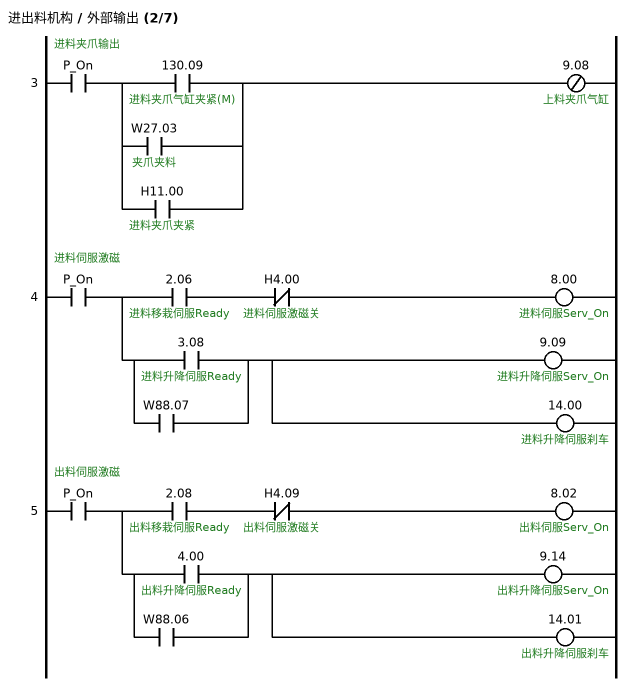
; [picture p120: 进出料机构 / 外部输出, rungs 3-5]
; rung 3: 进料夹爪输出
LD P_On
LD 130.09  ; 进料夹爪气缸夹紧(M)
OR W27.03  ; 夹爪夹料
OR H11.00  ; 进料夹爪夹紧
ANDLD
OUTNOT 9.08  ; 上料夹爪气缸
; rung 4: 进料伺服激磁
LD P_On
OUT TR0
AND 2.06  ; 进料移栽伺服Ready
ANDNOT H4.00  ; 进料伺服激磁关
OUT 8.00  ; 进料伺服Serv_On
LD TR0
LD 3.08  ; 进料升降伺服Ready
OR W88.07
ANDLD
OUT 9.09  ; 进料升降伺服Serv_On
OUT 14.00  ; 进料升降伺服刹车
; rung 5: 出料伺服激磁
LD P_On
OUT TR0
AND 2.08  ; 出料移栽伺服Ready
ANDNOT H4.09  ; 出料伺服激磁关
OUT 8.02  ; 出料伺服Serv_On
LD TR0
LD 4.00  ; 出料升降伺服Ready
OR W88.06
ANDLD
OUT 9.14  ; 出料升降伺服Serv_On
OUT 14.01  ; 出料升降伺服刹车

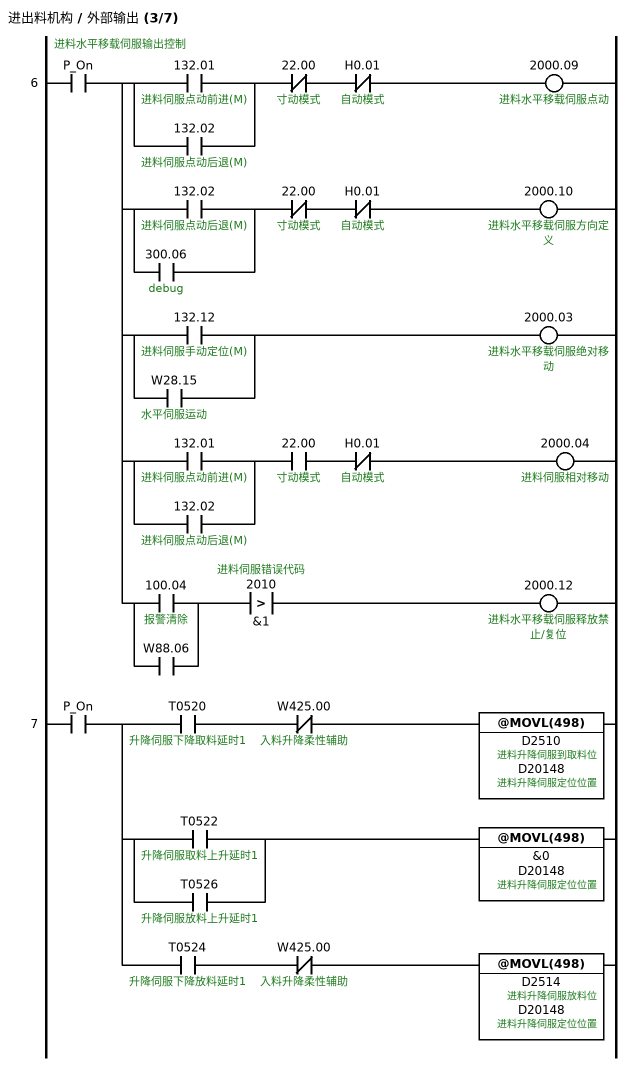
; rung 6: 进料水平移载伺服输出控制
LD P_On
OUT TR0
LD 132.01  ; 进料伺服点动前进(M)
OR 132.02  ; 进料伺服点动后退(M)
ANDLD
ANDNOT 22.00  ; 寸动模式
ANDNOT H0.01  ; 自动模式
OUT 2000.09  ; 进料水平移载伺服点动
LD TR0
LD 132.02  ; 进料伺服点动后退(M)
OR 300.06  ; debug
ANDLD
ANDNOT 22.00  ; 寸动模式
ANDNOT H0.01  ; 自动模式
OUT 2000.10  ; 进料水平移载伺服方向定义
LD TR0
LD 132.12  ; 进料伺服手动定位(M)
OR W28.15  ; 水平伺服运动
ANDLD
OUT 2000.03  ; 进料水平移载伺服绝对移动
LD TR0
LD 132.01  ; 进料伺服点动前进(M)
OR 132.02  ; 进料伺服点动后退(M)
ANDLD
AND 22.00  ; 寸动模式
ANDNOT H0.01  ; 自动模式
OUT 2000.04  ; 进料伺服相对移动
LD TR0
LD 100.04  ; 报警清除
OR W88.06
ANDLD
AND>(320) 2010 &1  ; 进料伺服错误代码
OUT 2000.12  ; 进料水平移载伺服释放禁止/复位
; rung 7
LD P_On
OUT TR0
AND T0520  ; 升降伺服下降取料延时1
ANDNOT W425.00  ; 入料升降柔性辅助
@MOVL(498) D2510 D20148  ; 进料升降伺服到取料位, 进料升降伺服定位位置
LD TR0
LD T0522  ; 升降伺服取料上升延时1
OR T0526  ; 升降伺服放料上升延时1
ANDLD
@MOVL(498) &0 D20148  ; 进料升降伺服定位位置
LD TR0
AND T0524  ; 升降伺服下降放料延时1
ANDNOT W425.00  ; 入料升降柔性辅助
@MOVL(498) D2514 D20148  ; 进料升降伺服放料位, 进料升降伺服定位位置

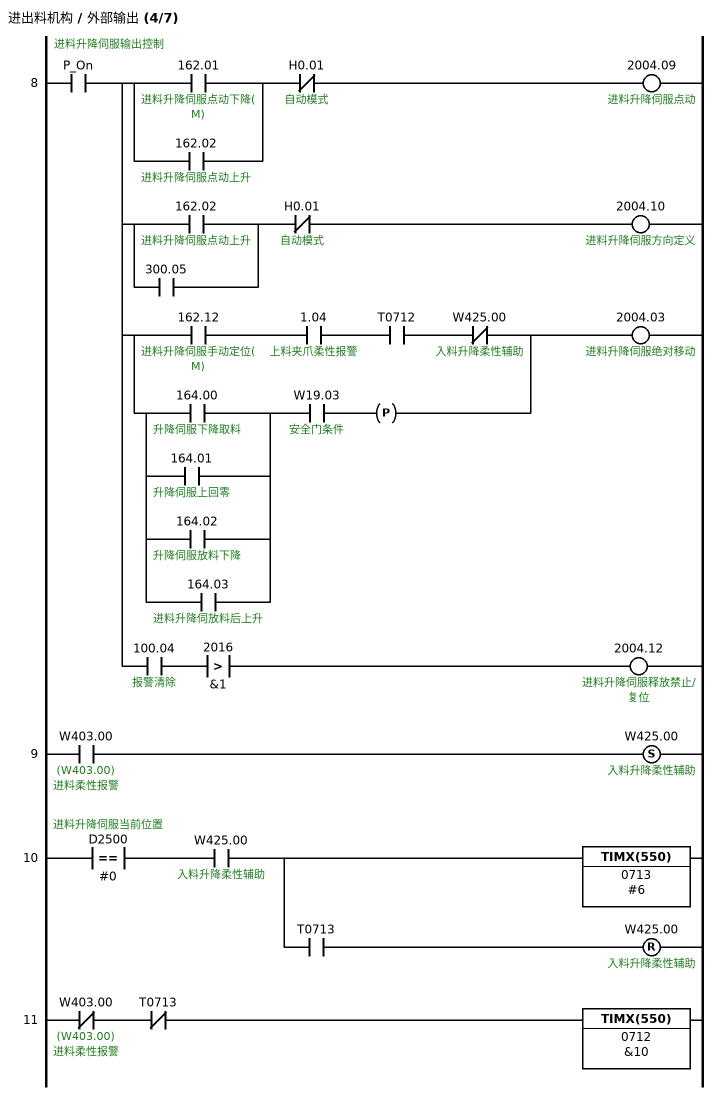
; rung 8: 进料升降伺服输出控制
LD P_On
OUT TR0
LD 162.01  ; 进料升降伺服点动下降(M)
OR 162.02  ; 进料升降伺服点动上升
ANDLD
ANDNOT H0.01  ; 自动模式
OUT 2004.09  ; 进料升降伺服点动
LD TR0
LD 162.02  ; 进料升降伺服点动上升
OR 300.05
ANDLD
ANDNOT H0.01  ; 自动模式
OUT 2004.10  ; 进料升降伺服方向定义
LD TR0
LD 162.12  ; 进料升降伺服手动定位(M)
AND 1.04  ; 上料夹爪柔性报警
AND T0712
ANDNOT W425.00  ; 入料升降柔性辅助
LD 164.00  ; 升降伺服下降取料
OR 164.01  ; 升降伺服上回零
OR 164.02  ; 升降伺服放料下降
OR 164.03  ; 进料升降伺放料后上升
AND W19.03  ; 安全门条件
UP(521)
ORLD
ANDLD
OUT 2004.03  ; 进料升降伺服绝对移动
LD TR0
AND 100.04  ; 报警清除
AND>(320) 2016 &1
OUT 2004.12  ; 进料升降伺服释放禁止/复位
; rung 9
LD W403.00  ; (W403.00) 进料柔性报警
SET W425.00  ; 入料升降柔性辅助
; rung 10
LD=L(301) D2500 #0  ; 进料升降伺服当前位置
AND W425.00  ; 入料升降柔性辅助
TIMX(550) 0713 #6
AND T0713
RSET W425.00  ; 入料升降柔性辅助
; rung 11
LDNOT W403.00  ; (W403.00) 进料柔性报警
ANDNOT T0713
TIMX(550) 0712 &10

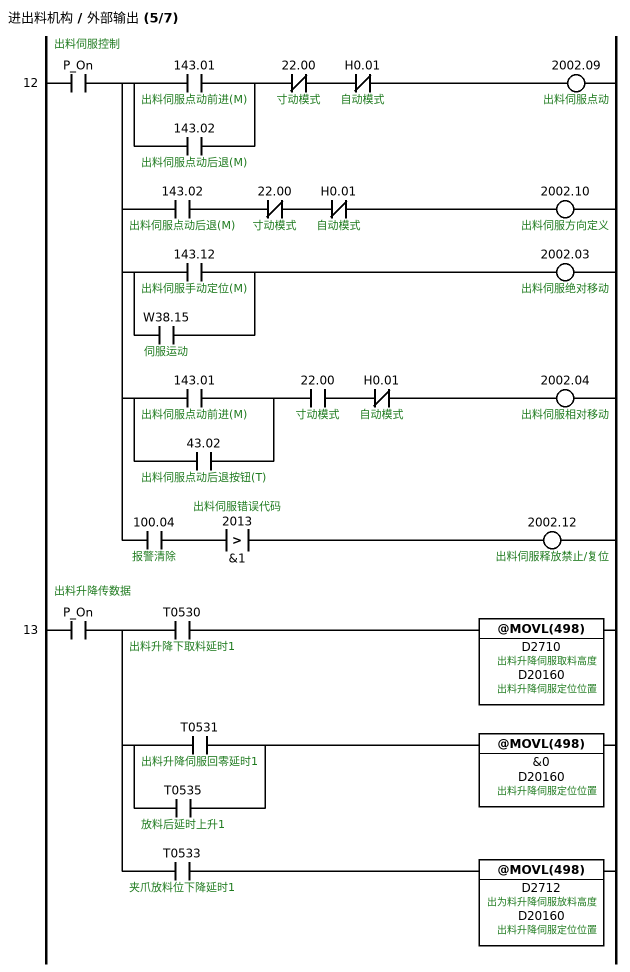
; rung 12: 出料伺服控制
LD P_On
OUT TR0
LD 143.01  ; 出料伺服点动前进(M)
OR 143.02  ; 出料伺服点动后退(M)
ANDLD
ANDNOT 22.00  ; 寸动模式
ANDNOT H0.01  ; 自动模式
OUT 2002.09  ; 出料伺服点动
LD TR0
AND 143.02  ; 出料伺服点动后退(M)
ANDNOT 22.00  ; 寸动模式
ANDNOT H0.01  ; 自动模式
OUT 2002.10  ; 出料伺服方向定义
LD TR0
LD 143.12  ; 出料伺服手动定位(M)
OR W38.15  ; 伺服运动
ANDLD
OUT 2002.03  ; 出料伺服绝对移动
LD TR0
LD 143.01  ; 出料伺服点动前进(M)
OR 43.02  ; 出料伺服点动后退按钮(T)
ANDLD
AND 22.00  ; 寸动模式
ANDNOT H0.01  ; 自动模式
OUT 2002.04  ; 出料伺服相对移动
LD TR0
AND 100.04  ; 报警清除
AND>(320) 2013 &1  ; 出料伺服错误代码
OUT 2002.12  ; 出料伺服释放禁止/复位
; rung 13: 出料升降传数据
LD P_On
OUT TR0
AND T0530  ; 出料升降下取料延时1
@MOVL(498) D2710 D20160  ; 出料升降伺服取料高度, 出料升降伺服定位位置
LD TR0
LD T0531  ; 出料升降伺服回零延时1
OR T0535  ; 放料后延时上升1
ANDLD
@MOVL(498) &0 D20160  ; 出料升降伺服定位位置
LD TR0
AND T0533  ; 夹爪放料位下降延时1
@MOVL(498) D2712 D20160  ; 出为料升降伺服放料高度, 出料升降伺服定位位置

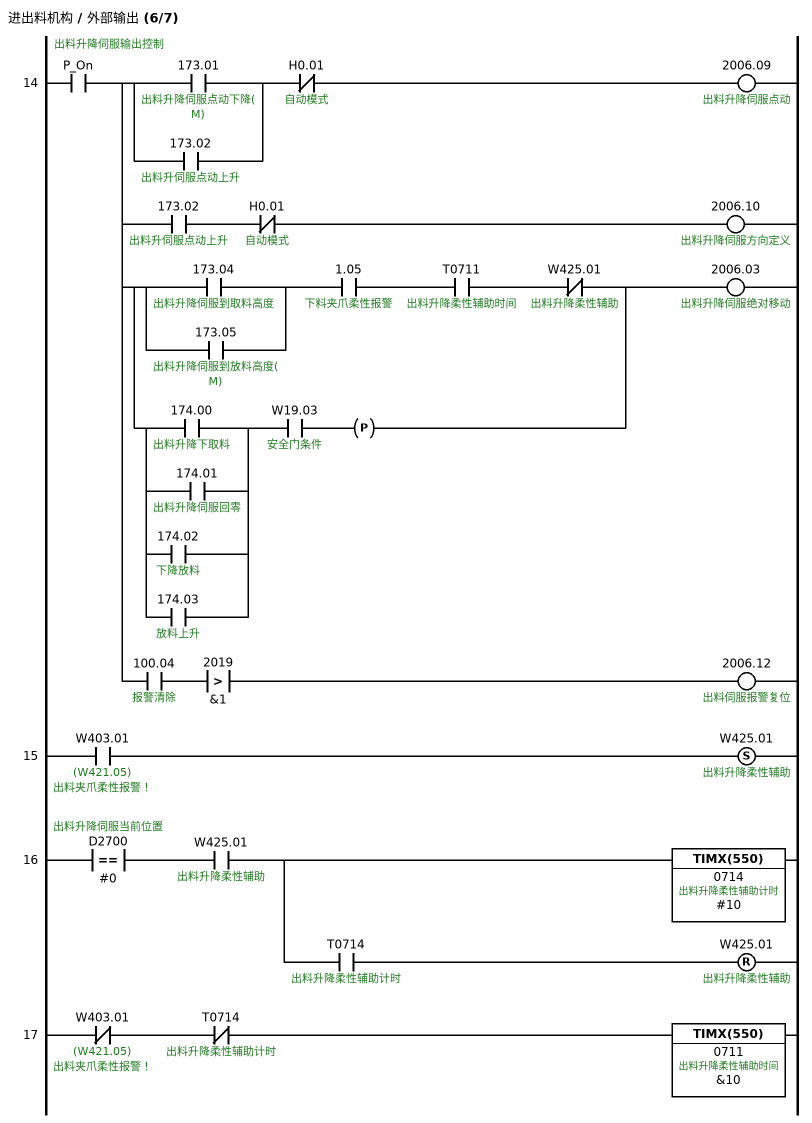
; rung 14: 出料升降伺服输出控制
LD P_On
OUT TR0
LD 173.01  ; 出料升降伺服点动下降(M)
OR 173.02  ; 出料升伺服点动上升
ANDLD
ANDNOT H0.01  ; 自动模式
OUT 2006.09  ; 出料升降伺服点动
LD TR0
AND 173.02  ; 出料升伺服点动上升
ANDNOT H0.01  ; 自动模式
OUT 2006.10  ; 出料升降伺服方向定义
LD TR0
LD 173.04  ; 出料升降伺服到取料高度
OR 173.05  ; 出料升降伺服到放料高度(M)
AND 1.05  ; 下料夹爪柔性报警
AND T0711  ; 出料升降柔性辅助时间
ANDNOT W425.01  ; 出料升降柔性辅助
LD 174.00  ; 出料升降下取料
OR 174.01  ; 出料升降伺服回零
OR 174.02  ; 下降放料
OR 174.03  ; 放料上升
AND W19.03  ; 安全门条件
UP(521)
ORLD
ANDLD
OUT 2006.03  ; 出料升降伺服绝对移动
LD TR0
AND 100.04  ; 报警清除
AND>(320) 2019 &1
OUT 2006.12  ; 出料伺服报警复位
; rung 15
LD W403.01  ; (W421.05) 出料夹爪柔性报警！
SET W425.01  ; 出料升降柔性辅助
; rung 16
LD=L(301) D2700 #0  ; 出料升降伺服当前位置
AND W425.01  ; 出料升降柔性辅助
TIMX(550) 0714 #10  ; 出料升降柔性辅助计时
AND T0714  ; 出料升降柔性辅助计时
RSET W425.01  ; 出料升降柔性辅助
; rung 17
LDNOT W403.01  ; (W421.05) 出料夹爪柔性报警！
ANDNOT T0714  ; 出料升降柔性辅助计时
TIMX(550) 0711 &10  ; 出料升降柔性辅助时间

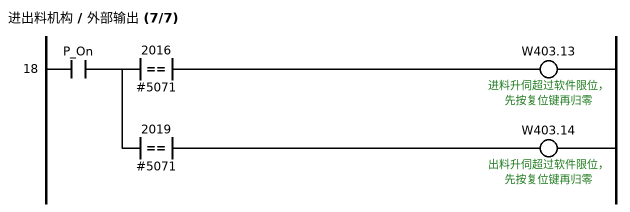
; rung 18
LD P_On
OUT TR0
AND=(300) 2016 #5071
OUT W403.13  ; 进料升伺超过软件限位，先按复位键再归零
LD TR0
AND=(300) 2019 #5071
OUT W403.14  ; 出料升伺超过软件限位，先按复位键再归零

### Section 指示灯

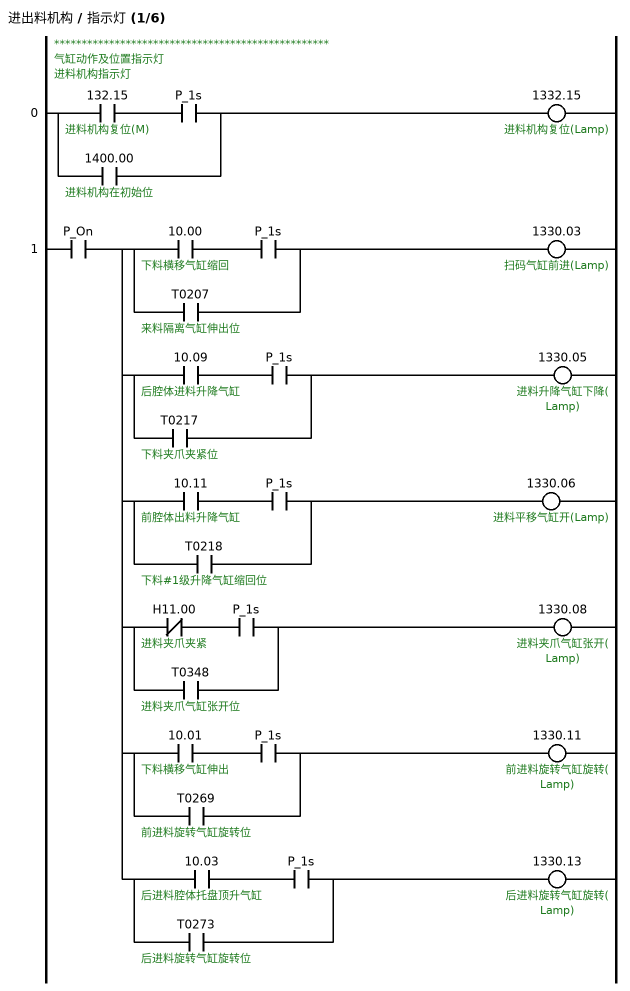
; rung 0: ************************************************** / 气缸动作及位置指示灯 / 进料机构指示灯
LD 132.15  ; 进料机构复位(M)
AND P_1s
OR 1400.00  ; 进料机构在初始位
OUT 1332.15  ; 进料机构复位(Lamp)
; rung 1
LD P_On
OUT TR0
LD 10.00  ; 下料横移气缸缩回
AND P_1s
OR T0207  ; 来料隔离气缸伸出位
ANDLD
OUT 1330.03  ; 扫码气缸前进(Lamp)
LD TR0
LD 10.09  ; 后腔体进料升降气缸
AND P_1s
OR T0217  ; 下料夹爪夹紧位
ANDLD
OUT 1330.05  ; 进料升降气缸下降(Lamp)
LD TR0
LD 10.11  ; 前腔体出料升降气缸
AND P_1s
OR T0218  ; 下料#1级升降气缸缩回位
ANDLD
OUT 1330.06  ; 进料平移气缸开(Lamp)
LD TR0
LDNOT H11.00  ; 进料夹爪夹紧
AND P_1s
OR T0348  ; 进料夹爪气缸张开位
ANDLD
OUT 1330.08  ; 进料夹爪气缸张开(Lamp)
LD TR0
LD 10.01  ; 下料横移气缸伸出
AND P_1s
OR T0269  ; 前进料旋转气缸旋转位
ANDLD
OUT 1330.11  ; 前进料旋转气缸旋转(Lamp)
LD TR0
LD 10.03  ; 后进料腔体托盘顶升气缸
AND P_1s
OR T0273  ; 后进料旋转气缸旋转位
ANDLD
OUT 1330.13  ; 后进料旋转气缸旋转(Lamp)

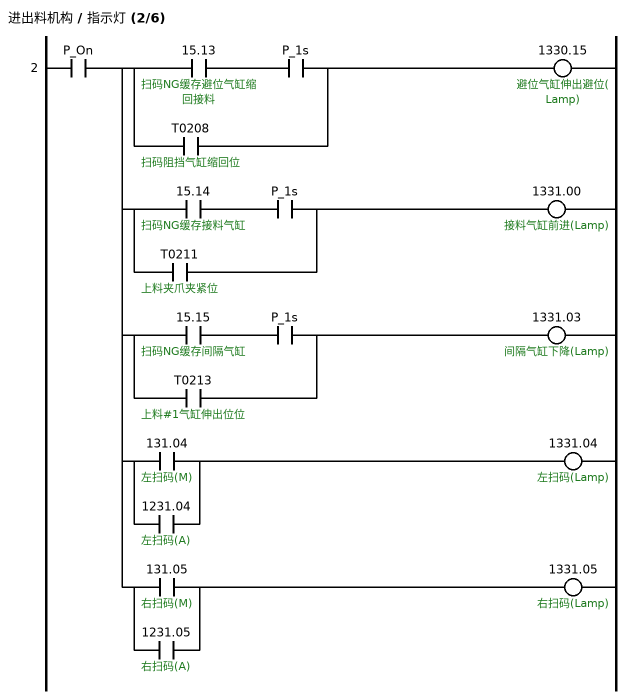
; rung 2
LD P_On
OUT TR0
LD 15.13  ; 扫码NG缓存避位气缸缩回接料
AND P_1s
OR T0208  ; 扫码阻挡气缸缩回位
ANDLD
OUT 1330.15  ; 避位气缸伸出避位(Lamp)
LD TR0
LD 15.14  ; 扫码NG缓存接料气缸
AND P_1s
OR T0211  ; 上料夹爪夹紧位
ANDLD
OUT 1331.00  ; 接料气缸前进(Lamp)
LD TR0
LD 15.15  ; 扫码NG缓存间隔气缸
AND P_1s
OR T0213  ; 上料#1气缸伸出位位
ANDLD
OUT 1331.03  ; 间隔气缸下降(Lamp)
LD TR0
LD 131.04  ; 左扫码(M)
OR 1231.04  ; 左扫码(A)
ANDLD
OUT 1331.04  ; 左扫码(Lamp)
LD TR0
LD 131.05  ; 右扫码(M)
OR 1231.05  ; 右扫码(A)
ANDLD
OUT 1331.05  ; 右扫码(Lamp)

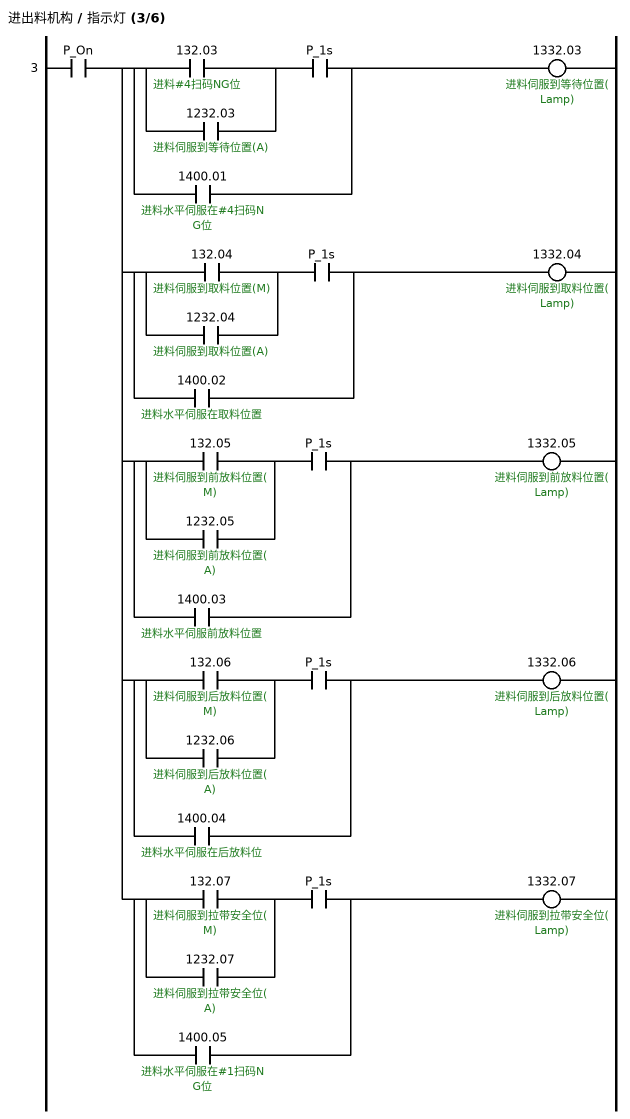
; rung 3
LD P_On
OUT TR0
LD 132.03  ; 进料#4扫码NG位
OR 1232.03  ; 进料伺服到等待位置(A)
AND P_1s
OR 1400.01  ; 进料水平伺服在#4扫码NG位
ANDLD
OUT 1332.03  ; 进料伺服到等待位置(Lamp)
LD TR0
LD 132.04  ; 进料伺服到取料位置(M)
OR 1232.04  ; 进料伺服到取料位置(A)
AND P_1s
OR 1400.02  ; 进料水平伺服在取料位置
ANDLD
OUT 1332.04  ; 进料伺服到取料位置(Lamp)
LD TR0
LD 132.05  ; 进料伺服到前放料位置(M)
OR 1232.05  ; 进料伺服到前放料位置(A)
AND P_1s
OR 1400.03  ; 进料水平伺服前放料位置
ANDLD
OUT 1332.05  ; 进料伺服到前放料位置(Lamp)
LD TR0
LD 132.06  ; 进料伺服到后放料位置(M)
OR 1232.06  ; 进料伺服到后放料位置(A)
AND P_1s
OR 1400.04  ; 进料水平伺服在后放料位
ANDLD
OUT 1332.06  ; 进料伺服到后放料位置(Lamp)
LD TR0
LD 132.07  ; 进料伺服到拉带安全位(M)
OR 1232.07  ; 进料伺服到拉带安全位(A)
AND P_1s
OR 1400.05  ; 进料水平伺服在#1扫码NG位
ANDLD
OUT 1332.07  ; 进料伺服到拉带安全位(Lamp)

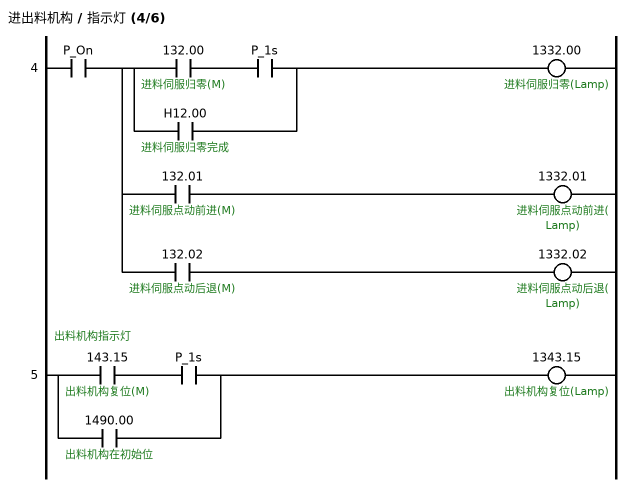
; rung 4
LD P_On
OUT TR0
LD 132.00  ; 进料伺服归零(M)
AND P_1s
OR H12.00  ; 进料伺服归零完成
ANDLD
OUT 1332.00  ; 进料伺服归零(Lamp)
LD TR0
AND 132.01  ; 进料伺服点动前进(M)
OUT 1332.01  ; 进料伺服点动前进(Lamp)
LD TR0
AND 132.02  ; 进料伺服点动后退(M)
OUT 1332.02  ; 进料伺服点动后退(Lamp)
; rung 5: 出料机构指示灯
LD 143.15  ; 出料机构复位(M)
AND P_1s
OR 1490.00  ; 出料机构在初始位
OUT 1343.15  ; 出料机构复位(Lamp)

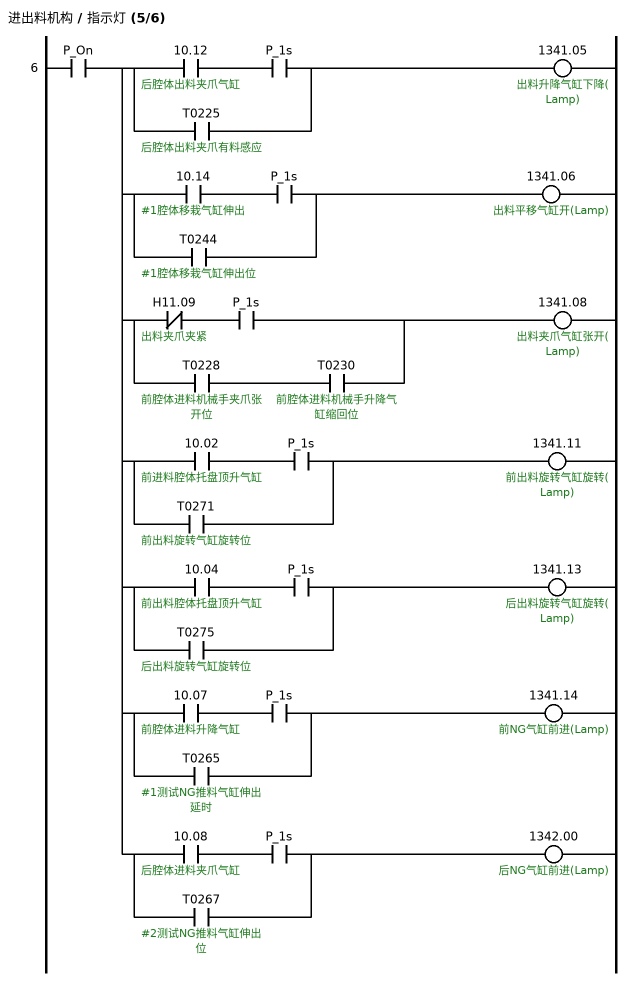
; rung 6
LD P_On
OUT TR0
LD 10.12  ; 后腔体出料夹爪气缸
AND P_1s
OR T0225  ; 后腔体出料夹爪有料感应
ANDLD
OUT 1341.05  ; 出料升降气缸下降(Lamp)
LD TR0
LD 10.14  ; #1腔体移栽气缸伸出
AND P_1s
OR T0244  ; #1腔体移栽气缸伸出位
ANDLD
OUT 1341.06  ; 出料平移气缸开(Lamp)
LD TR0
LDNOT H11.09  ; 出料夹爪夹紧
AND P_1s
LD T0228  ; 前腔体进料机械手夹爪张开位
AND T0230  ; 前腔体进料机械手升降气缸缩回位
ORLD
ANDLD
OUT 1341.08  ; 出料夹爪气缸张开(Lamp)
LD TR0
LD 10.02  ; 前进料腔体托盘顶升气缸
AND P_1s
OR T0271  ; 前出料旋转气缸旋转位
ANDLD
OUT 1341.11  ; 前出料旋转气缸旋转(Lamp)
LD TR0
LD 10.04  ; 前出料腔体托盘顶升气缸
AND P_1s
OR T0275  ; 后出料旋转气缸旋转位
ANDLD
OUT 1341.13  ; 后出料旋转气缸旋转(Lamp)
LD TR0
LD 10.07  ; 前腔体进料升降气缸
AND P_1s
OR T0265  ; #1测试NG推料气缸伸出延时
ANDLD
OUT 1341.14  ; 前NG气缸前进(Lamp)
LD TR0
LD 10.08  ; 后腔体进料夹爪气缸
AND P_1s
OR T0267  ; #2测试NG推料气缸伸出位
ANDLD
OUT 1342.00  ; 后NG气缸前进(Lamp)

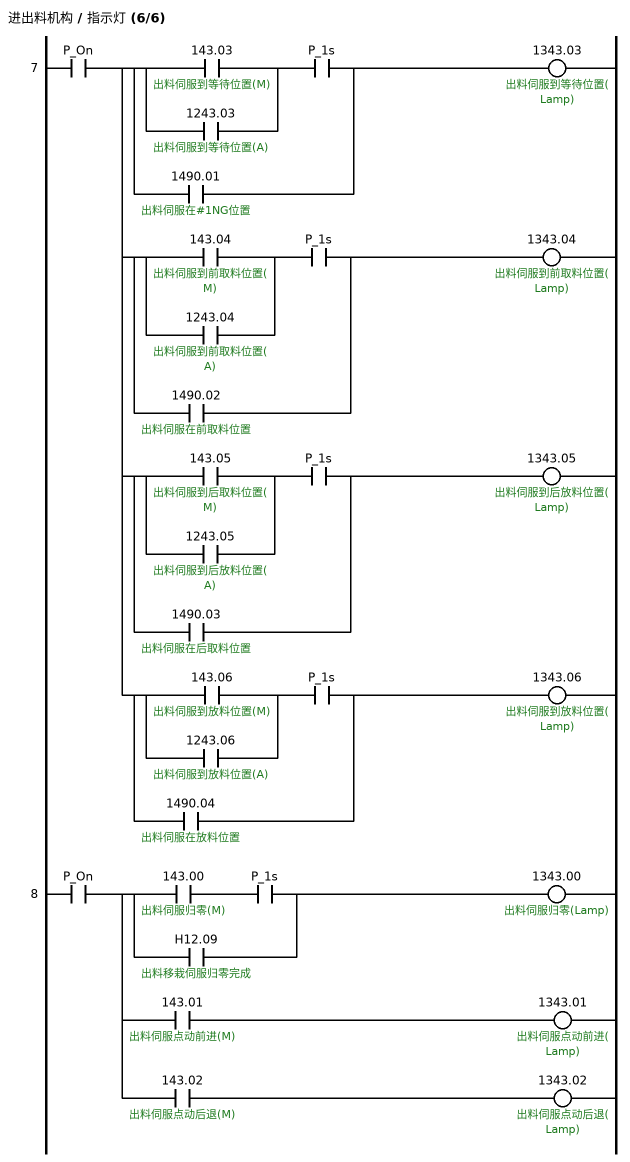
; rung 7
LD P_On
OUT TR0
LD 143.03  ; 出料伺服到等待位置(M)
OR 1243.03  ; 出料伺服到等待位置(A)
AND P_1s
OR 1490.01  ; 出料伺服在#1NG位置
ANDLD
OUT 1343.03  ; 出料伺服到等待位置(Lamp)
LD TR0
LD 143.04  ; 出料伺服到前取料位置(M)
OR 1243.04  ; 出料伺服到前取料位置(A)
AND P_1s
OR 1490.02  ; 出料伺服在前取料位置
ANDLD
OUT 1343.04  ; 出料伺服到前取料位置(Lamp)
LD TR0
LD 143.05  ; 出料伺服到后取料位置(M)
OR 1243.05  ; 出料伺服到后放料位置(A)
AND P_1s
OR 1490.03  ; 出料伺服在后取料位置
ANDLD
OUT 1343.05  ; 出料伺服到后放料位置(Lamp)
LD TR0
LD 143.06  ; 出料伺服到放料位置(M)
OR 1243.06  ; 出料伺服到放料位置(A)
AND P_1s
OR 1490.04  ; 出料伺服在放料位置
ANDLD
OUT 1343.06  ; 出料伺服到放料位置(Lamp)
; rung 8
LD P_On
OUT TR0
LD 143.00  ; 出料伺服归零(M)
AND P_1s
OR H12.09  ; 出料移栽伺服归零完成
ANDLD
OUT 1343.00  ; 出料伺服归零(Lamp)
LD TR0
AND 143.01  ; 出料伺服点动前进(M)
OUT 1343.01  ; 出料伺服点动前进(Lamp)
LD TR0
AND 143.02  ; 出料伺服点动后退(M)
OUT 1343.02  ; 出料伺服点动后退(Lamp)

### Section END
; rung 0
END(001)

## Program 前上料机构 (cyclic task 2)

### Section Main

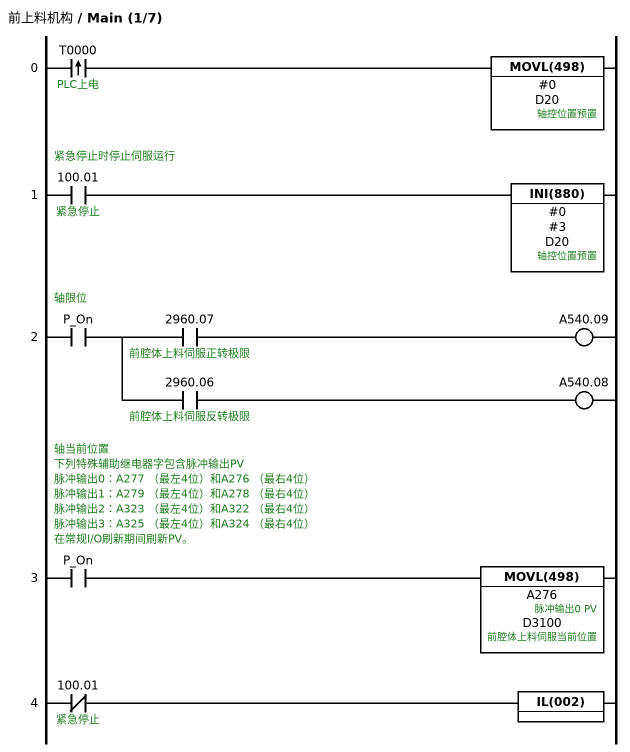
; rung 0
@LD T0000  ; PLC上电
MOVL(498) #0 D20  ; 轴控位置预置
; rung 1: 紧急停止时停止伺服运行
LD 100.01  ; 紧急停止
INI(880) #0 #3 D20  ; 轴控位置预置
; rung 2: 轴限位
LD P_On
OUT TR0
AND 2960.07  ; 前腔体上料伺服正转极限
OUT A540.09
LD TR0
AND 2960.06  ; 前腔体上料伺服反转极限
OUT A540.08
; rung 3: 轴当前位置 / 下列特殊辅助继电器字包含脉冲输出PV / 脉冲输出0：A277 （最左4位）和A276 （最右4位） / 脉冲输出1：A279 （最左4位）和A278 （最右4位） / 脉冲输出2：A323 （最左4位）和A322 （最右4位） / 脉冲输出3：A325 （最左4位）和A324 （最右4位） / 在常规I/O刷新期间刷新PV。
LD P_On
MOVL(498) A276 D3100  ; 脉冲输出0 PV, 前腔体上料伺服当前位置
; rung 4
LDNOT 100.01  ; 紧急停止
IL(002)

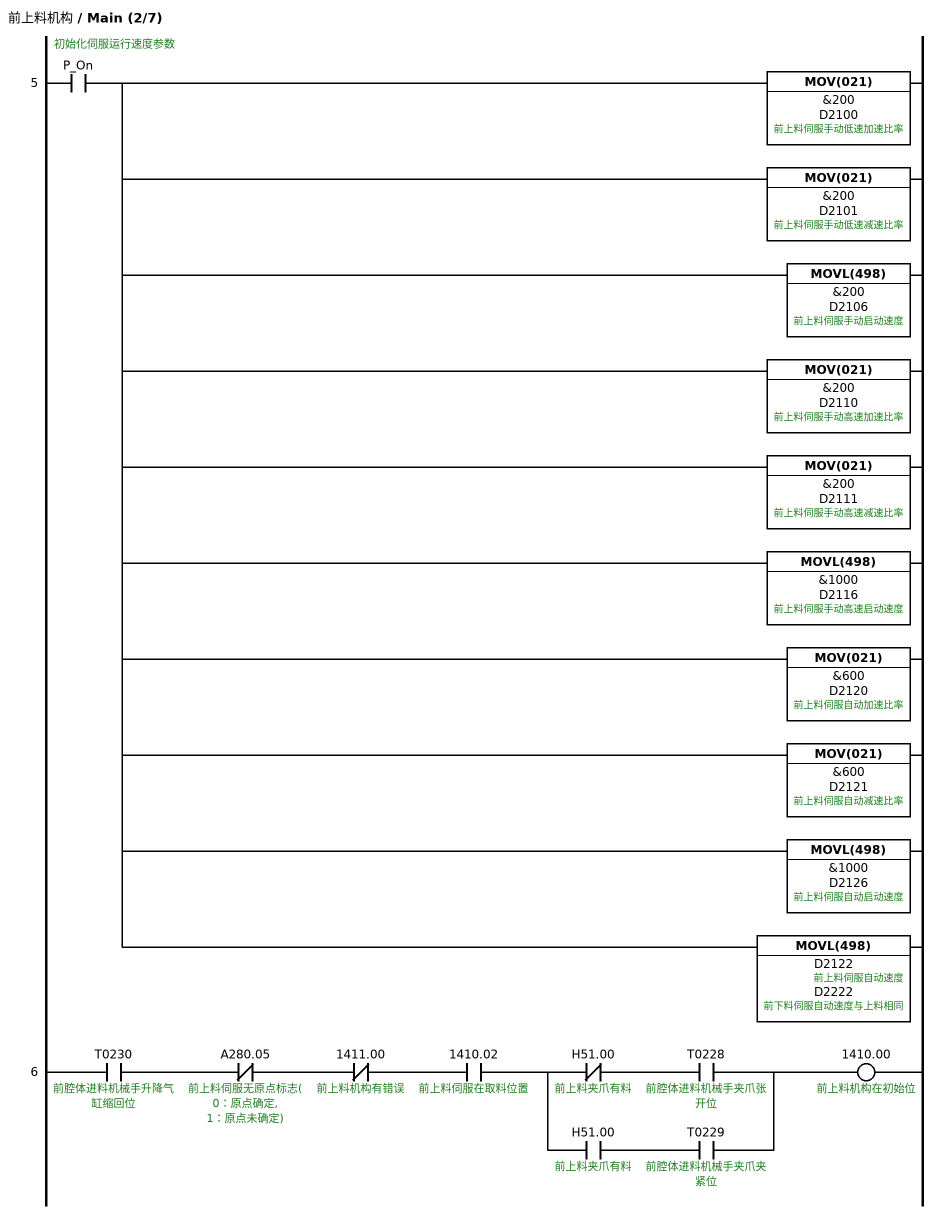
; rung 5: 初始化伺服运行速度参数
LD P_On
MOV(021) &200 D2100  ; 前上料伺服手动低速加速比率
MOV(021) &200 D2101  ; 前上料伺服手动低速减速比率
MOVL(498) &200 D2106  ; 前上料伺服手动启动速度
MOV(021) &200 D2110  ; 前上料伺服手动高速加速比率
MOV(021) &200 D2111  ; 前上料伺服手动高速减速比率
MOVL(498) &1000 D2116  ; 前上料伺服手动高速启动速度
MOV(021) &600 D2120  ; 前上料伺服自动加速比率
MOV(021) &600 D2121  ; 前上料伺服自动减速比率
MOVL(498) &1000 D2126  ; 前上料伺服自动启动速度
MOVL(498) D2122 D2222  ; 前上料伺服自动速度, 前下料伺服自动速度与上料相同
; rung 6
LD T0230  ; 前腔体进料机械手升降气缸缩回位
ANDNOT A280.05  ; 前上料伺服无原点标志(0：原点确定,1：原点未确定)
ANDNOT 1411.00  ; 前上料机构有错误
AND 1410.02  ; 前上料伺服在取料位置
LDNOT H51.00  ; 前上料夹爪有料
AND T0228  ; 前腔体进料机械手夹爪张开位
LD H51.00  ; 前上料夹爪有料
AND T0229  ; 前腔体进料机械手夹爪夹紧位
ORLD
ANDLD
OUT 1410.00  ; 前上料机构在初始位

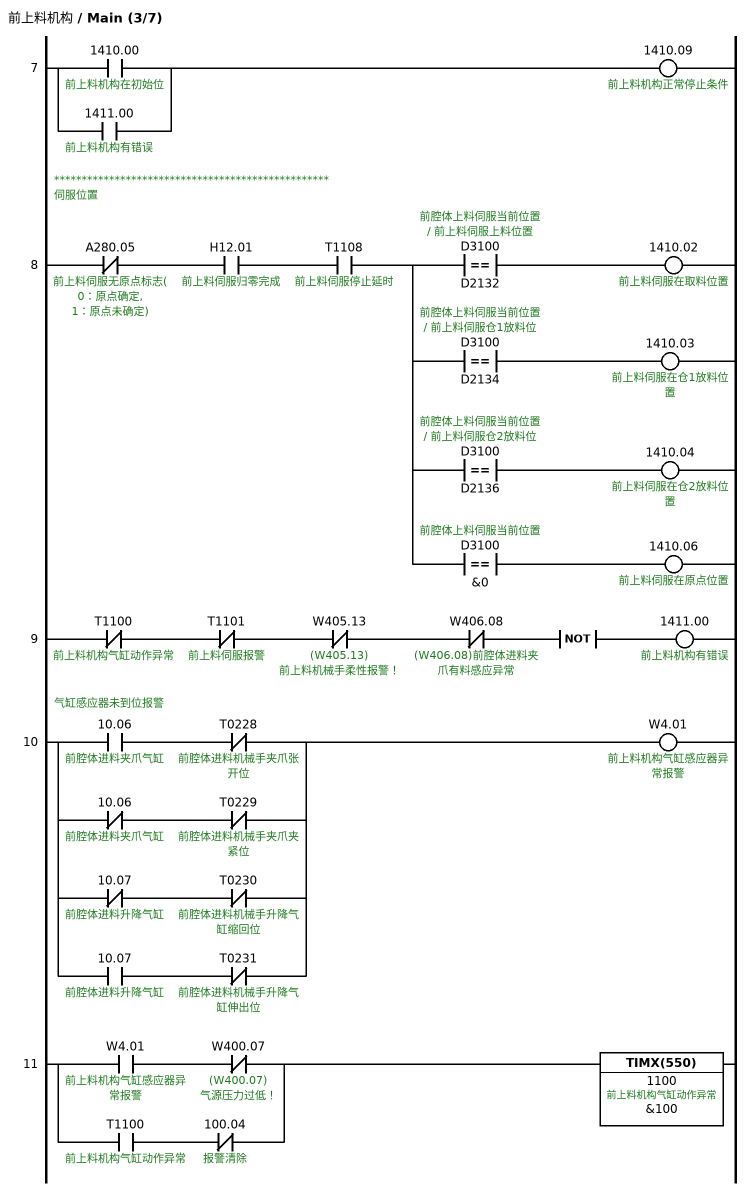
; rung 7
LD 1410.00  ; 前上料机构在初始位
OR 1411.00  ; 前上料机构有错误
OUT 1410.09  ; 前上料机构正常停止条件
; rung 8: ************************************************** / 伺服位置
LDNOT A280.05  ; 前上料伺服无原点标志(0：原点确定,1：原点未确定)
AND H12.01  ; 前上料伺服归零完成
AND T1108  ; 前上料伺服停止延时
OUT TR0
AND=SL(303) D3100 D2132  ; 前腔体上料伺服当前位置, 前上料伺服上料位置
OUT 1410.02  ; 前上料伺服在取料位置
LD TR0
AND=SL(303) D3100 D2134  ; 前腔体上料伺服当前位置, 前上料伺服仓1放料位
OUT 1410.03  ; 前上料伺服在仓1放料位置
LD TR0
AND=SL(303) D3100 D2136  ; 前腔体上料伺服当前位置, 前上料伺服仓2放料位
OUT 1410.04  ; 前上料伺服在仓2放料位置
LD TR0
AND=SL(303) D3100 &0  ; 前腔体上料伺服当前位置
OUT 1410.06  ; 前上料伺服在原点位置
; rung 9
LDNOT T1100  ; 前上料机构气缸动作异常
ANDNOT T1101  ; 前上料伺服报警
ANDNOT W405.13  ; (W405.13) 前上料机械手柔性报警！
ANDNOT W406.08  ; (W406.08)前腔体进料夹爪有料感应异常
NOT(520)
OUT 1411.00  ; 前上料机构有错误
; rung 10: 气缸感应器未到位报警
LD 10.06  ; 前腔体进料夹爪气缸
ANDNOT T0228  ; 前腔体进料机械手夹爪张开位
LDNOT 10.06  ; 前腔体进料夹爪气缸
ANDNOT T0229  ; 前腔体进料机械手夹爪夹紧位
ORLD
LDNOT 10.07  ; 前腔体进料升降气缸
ANDNOT T0230  ; 前腔体进料机械手升降气缸缩回位
ORLD
LD 10.07  ; 前腔体进料升降气缸
ANDNOT T0231  ; 前腔体进料机械手升降气缸伸出位
ORLD
OUT W4.01  ; 前上料机构气缸感应器异常报警
; rung 11
LD W4.01  ; 前上料机构气缸感应器异常报警
ANDNOT W400.07  ; (W400.07) 气源压力过低！
LD T1100  ; 前上料机构气缸动作异常
ANDNOT 100.04  ; 报警清除
ORLD
TIMX(550) 1100 &100  ; 前上料机构气缸动作异常

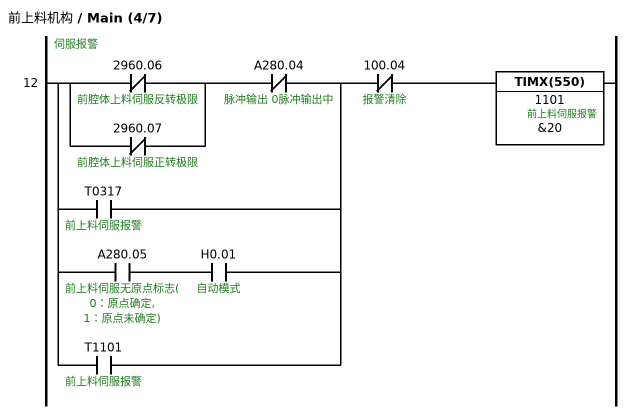
; rung 12: 伺服报警
LDNOT 2960.06  ; 前腔体上料伺服反转极限
ORNOT 2960.07  ; 前腔体上料伺服正转极限
ANDNOT A280.04  ; 脉冲输出 0脉冲输出中
OR T0317  ; 前上料伺服报警
LD A280.05  ; 前上料伺服无原点标志(0：原点确定,1：原点未确定)
AND H0.01  ; 自动模式
ORLD
OR T1101  ; 前上料伺服报警
ANDNOT 100.04  ; 报警清除
TIMX(550) 1101 &20  ; 前上料伺服报警

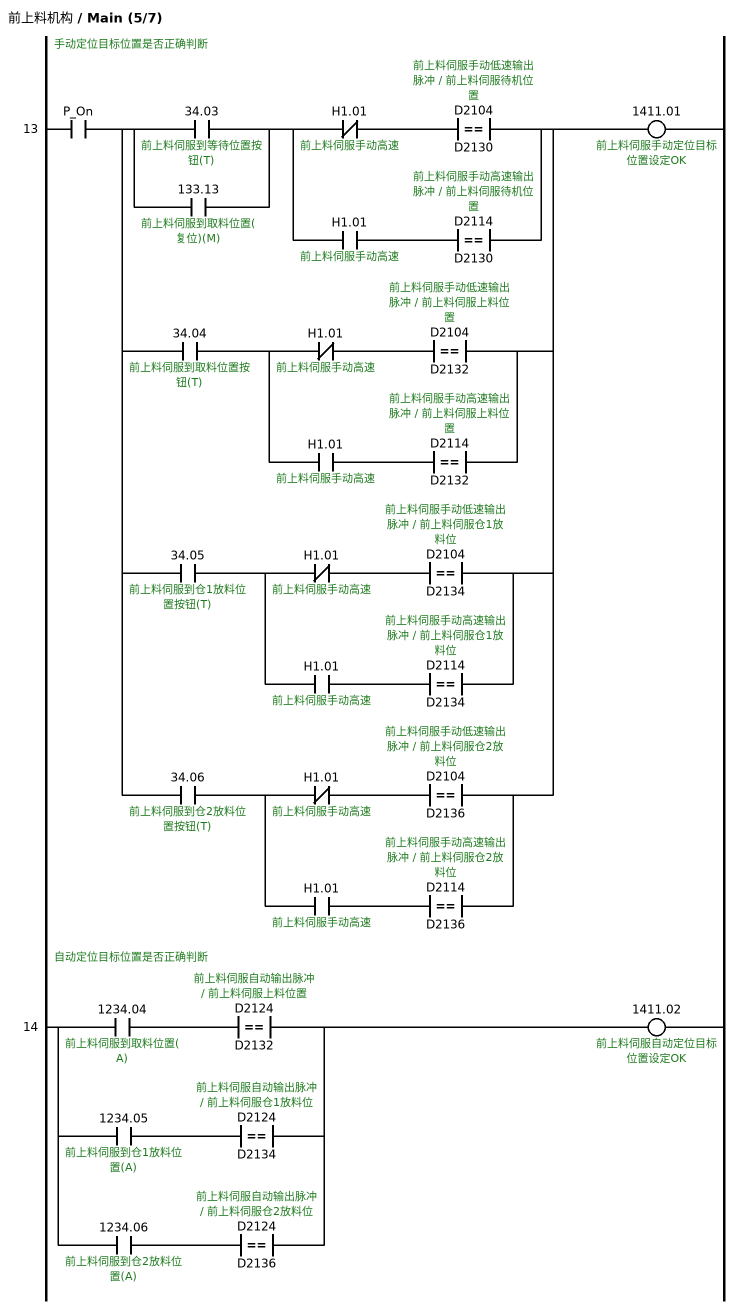
; rung 13: 手动定位目标位置是否正确判断
LD P_On
LD 34.03  ; 前上料伺服到等待位置按钮(T)
OR 133.13  ; 前上料伺服到取料位置(复位)(M)
LDNOT H1.01  ; 前上料伺服手动高速
AND=SL(303) D2104 D2130  ; 前上料伺服手动低速输出脉冲, 前上料伺服待机位置
LD H1.01  ; 前上料伺服手动高速
AND=SL(303) D2114 D2130  ; 前上料伺服手动高速输出脉冲, 前上料伺服待机位置
ORLD
ANDLD
LD 34.04  ; 前上料伺服到取料位置按钮(T)
LDNOT H1.01  ; 前上料伺服手动高速
AND=SL(303) D2104 D2132  ; 前上料伺服手动低速输出脉冲, 前上料伺服上料位置
LD H1.01  ; 前上料伺服手动高速
AND=SL(303) D2114 D2132  ; 前上料伺服手动高速输出脉冲, 前上料伺服上料位置
ORLD
ANDLD
ORLD
LD 34.05  ; 前上料伺服到仓1放料位置按钮(T)
LDNOT H1.01  ; 前上料伺服手动高速
AND=SL(303) D2104 D2134  ; 前上料伺服手动低速输出脉冲, 前上料伺服仓1放料位
LD H1.01  ; 前上料伺服手动高速
AND=SL(303) D2114 D2134  ; 前上料伺服手动高速输出脉冲, 前上料伺服仓1放料位
ORLD
ANDLD
ORLD
LD 34.06  ; 前上料伺服到仓2放料位置按钮(T)
LDNOT H1.01  ; 前上料伺服手动高速
AND=SL(303) D2104 D2136  ; 前上料伺服手动低速输出脉冲, 前上料伺服仓2放料位
LD H1.01  ; 前上料伺服手动高速
AND=SL(303) D2114 D2136  ; 前上料伺服手动高速输出脉冲, 前上料伺服仓2放料位
ORLD
ANDLD
ORLD
ANDLD
OUT 1411.01  ; 前上料伺服手动定位目标位置设定OK
; rung 14: 自动定位目标位置是否正确判断
LD 1234.04  ; 前上料伺服到取料位置(A)
AND=SL(303) D2124 D2132  ; 前上料伺服自动输出脉冲, 前上料伺服上料位置
LD 1234.05  ; 前上料伺服到仓1放料位置(A)
AND=SL(303) D2124 D2134  ; 前上料伺服自动输出脉冲, 前上料伺服仓1放料位
ORLD
LD 1234.06  ; 前上料伺服到仓2放料位置(A)
AND=SL(303) D2124 D2136  ; 前上料伺服自动输出脉冲, 前上料伺服仓2放料位
ORLD
OUT 1411.02  ; 前上料伺服自动定位目标位置设定OK

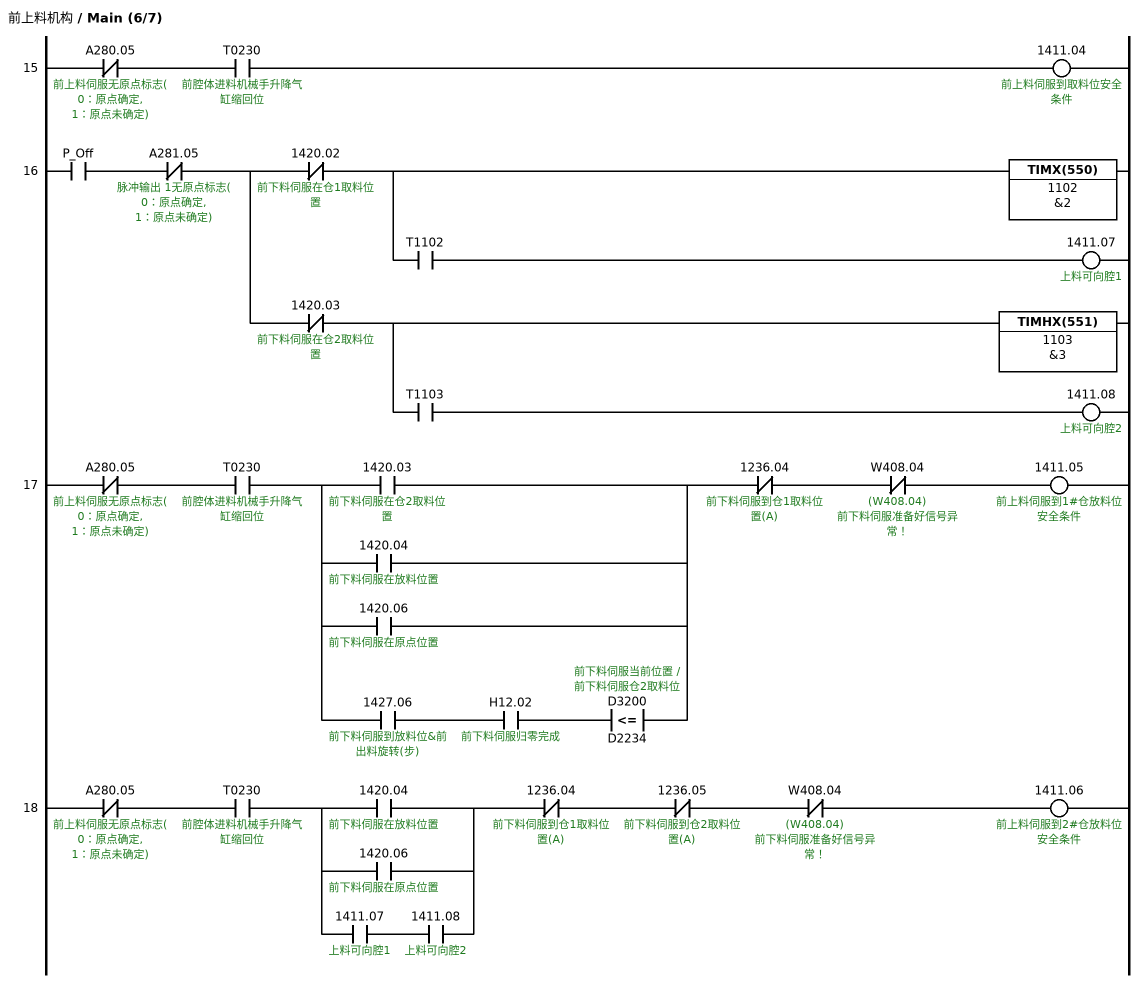
; rung 15
LDNOT A280.05  ; 前上料伺服无原点标志(0：原点确定,1：原点未确定)
AND T0230  ; 前腔体进料机械手升降气缸缩回位
OUT 1411.04  ; 前上料伺服到取料位安全条件
; rung 16
LD P_Off
ANDNOT A281.05  ; 脉冲输出 1无原点标志(0：原点确定,1：原点未确定)
OUT TR0
ANDNOT 1420.02  ; 前下料伺服在仓1取料位置
TIMX(550) 1102 &2
AND T1102
OUT 1411.07  ; 上料可向腔1
LD TR0
ANDNOT 1420.03  ; 前下料伺服在仓2取料位置
TIMHX(551) 1103 &3
AND T1103
OUT 1411.08  ; 上料可向腔2
; rung 17
LDNOT A280.05  ; 前上料伺服无原点标志(0：原点确定,1：原点未确定)
AND T0230  ; 前腔体进料机械手升降气缸缩回位
LD 1420.03  ; 前下料伺服在仓2取料位置
OR 1420.04  ; 前下料伺服在放料位置
OR 1420.06  ; 前下料伺服在原点位置
LD 1427.06  ; 前下料伺服到放料位&前出料旋转(步)
AND H12.02  ; 前下料伺服归零完成
AND<=SL(318) D3200 D2234  ; 前下料伺服当前位置, 前下料伺服仓2取料位
ORLD
ANDLD
ANDNOT 1236.04  ; 前下料伺服到仓1取料位置(A)
ANDNOT W408.04  ; (W408.04) 前下料伺服准备好信号异常！
OUT 1411.05  ; 前上料伺服到1#仓放料位安全条件
; rung 18
LDNOT A280.05  ; 前上料伺服无原点标志(0：原点确定,1：原点未确定)
AND T0230  ; 前腔体进料机械手升降气缸缩回位
LD 1420.04  ; 前下料伺服在放料位置
OR 1420.06  ; 前下料伺服在原点位置
LD 1411.07  ; 上料可向腔1
AND 1411.08  ; 上料可向腔2
ORLD
ANDLD
ANDNOT 1236.04  ; 前下料伺服到仓1取料位置(A)
ANDNOT 1236.05  ; 前下料伺服到仓2取料位置(A)
ANDNOT W408.04  ; (W408.04) 前下料伺服准备好信号异常！
OUT 1411.06  ; 前上料伺服到2#仓放料位安全条件

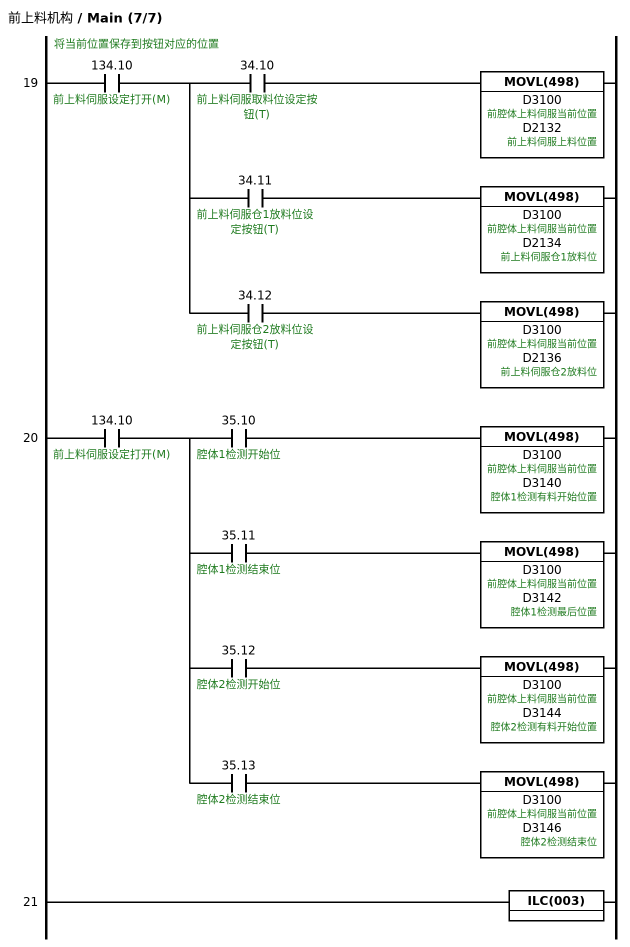
; rung 19: 将当前位置保存到按钮对应的位置
LD 134.10  ; 前上料伺服设定打开(M)
OUT TR0
AND 34.10  ; 前上料伺服取料位设定按钮(T)
MOVL(498) D3100 D2132  ; 前腔体上料伺服当前位置, 前上料伺服上料位置
LD TR0
AND 34.11  ; 前上料伺服仓1放料位设定按钮(T)
MOVL(498) D3100 D2134  ; 前腔体上料伺服当前位置, 前上料伺服仓1放料位
LD TR0
AND 34.12  ; 前上料伺服仓2放料位设定按钮(T)
MOVL(498) D3100 D2136  ; 前腔体上料伺服当前位置, 前上料伺服仓2放料位
; rung 20
LD 134.10  ; 前上料伺服设定打开(M)
OUT TR0
AND 35.10  ; 腔体1检测开始位
MOVL(498) D3100 D3140  ; 前腔体上料伺服当前位置, 腔体1检测有料开始位置
LD TR0
AND 35.11  ; 腔体1检测结束位
MOVL(498) D3100 D3142  ; 前腔体上料伺服当前位置, 腔体1检测最后位置
LD TR0
AND 35.12  ; 腔体2检测开始位
MOVL(498) D3100 D3144  ; 前腔体上料伺服当前位置, 腔体2检测有料开始位置
LD TR0
AND 35.13  ; 腔体2检测结束位
MOVL(498) D3100 D3146  ; 前腔体上料伺服当前位置, 腔体2检测结束位
; rung 21
ILC(003)

### Section 工站复位

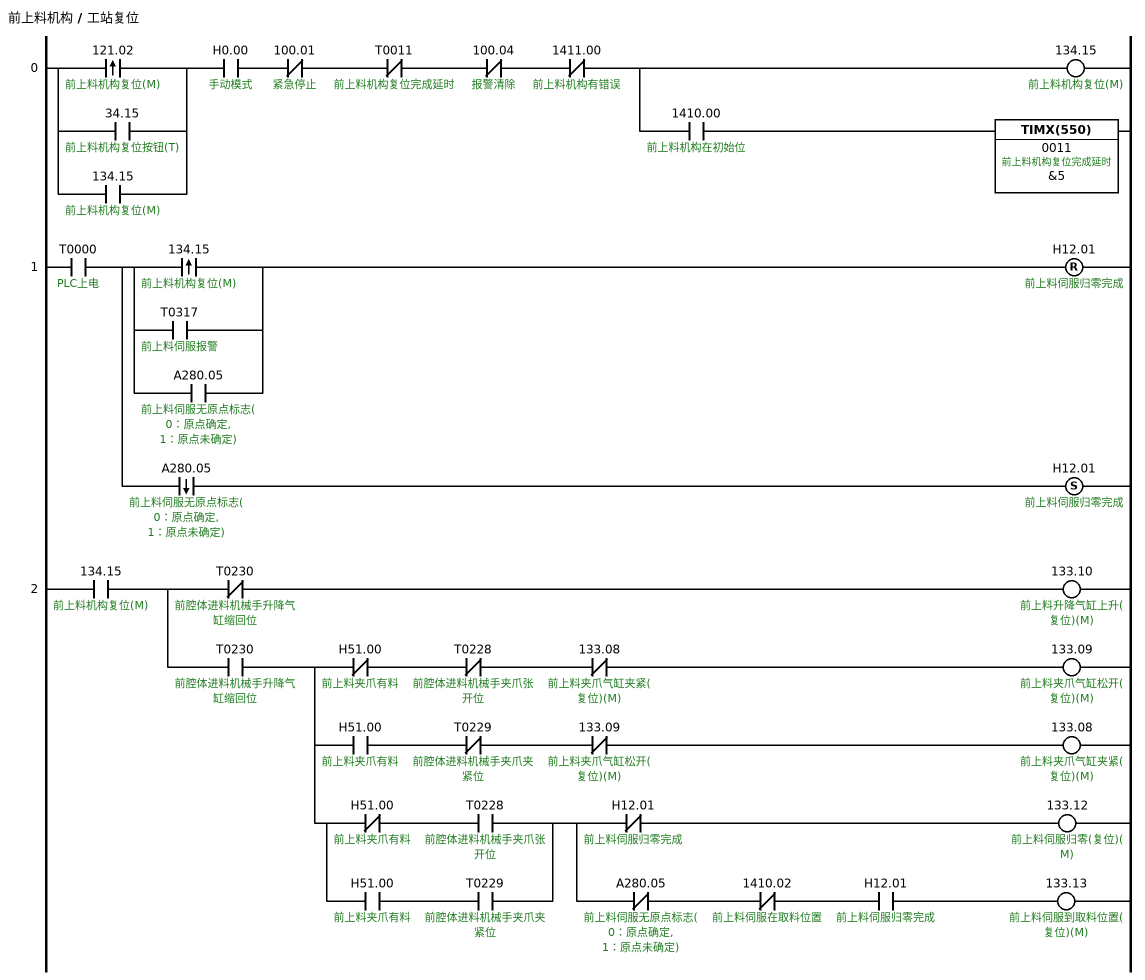
; rung 0
@LD 121.02  ; 前上料机构复位(M)
OR 34.15  ; 前上料机构复位按钮(T)
OR 134.15  ; 前上料机构复位(M)
AND H0.00  ; 手动模式
ANDNOT 100.01  ; 紧急停止
ANDNOT T0011  ; 前上料机构复位完成延时
ANDNOT 100.04  ; 报警清除
ANDNOT 1411.00  ; 前上料机构有错误
OUT 134.15  ; 前上料机构复位(M)
AND 1410.00  ; 前上料机构在初始位
TIMX(550) 0011 &5  ; 前上料机构复位完成延时
; rung 1
LD T0000  ; PLC上电
OUT TR0
@LD 134.15  ; 前上料机构复位(M)
OR T0317  ; 前上料伺服报警
OR A280.05  ; 前上料伺服无原点标志(0：原点确定,1：原点未确定)
ANDLD
RSET H12.01  ; 前上料伺服归零完成
LD TR0
%AND A280.05  ; 前上料伺服无原点标志(0：原点确定,1：原点未确定)
SET H12.01  ; 前上料伺服归零完成
; rung 2
LD 134.15  ; 前上料机构复位(M)
OUT TR0
ANDNOT T0230  ; 前腔体进料机械手升降气缸缩回位
OUT 133.10  ; 前上料升降气缸上升(复位)(M)
LD TR0
AND T0230  ; 前腔体进料机械手升降气缸缩回位
OUT TR0
ANDNOT H51.00  ; 前上料夹爪有料
ANDNOT T0228  ; 前腔体进料机械手夹爪张开位
ANDNOT 133.08  ; 前上料夹爪气缸夹紧(复位)(M)
OUT 133.09  ; 前上料夹爪气缸松开(复位)(M)
LD TR0
AND H51.00  ; 前上料夹爪有料
ANDNOT T0229  ; 前腔体进料机械手夹爪夹紧位
ANDNOT 133.09  ; 前上料夹爪气缸松开(复位)(M)
OUT 133.08  ; 前上料夹爪气缸夹紧(复位)(M)
LD TR0
LDNOT H51.00  ; 前上料夹爪有料
AND T0228  ; 前腔体进料机械手夹爪张开位
LD H51.00  ; 前上料夹爪有料
AND T0229  ; 前腔体进料机械手夹爪夹紧位
ORLD
ANDLD
OUT TR0
ANDNOT H12.01  ; 前上料伺服归零完成
OUT 133.12  ; 前上料伺服归零(复位)(M)
LD TR0
ANDNOT A280.05  ; 前上料伺服无原点标志(0：原点确定,1：原点未确定)
ANDNOT 1410.02  ; 前上料伺服在取料位置
AND H12.01  ; 前上料伺服归零完成
OUT 133.13  ; 前上料伺服到取料位置(复位)(M)

### Section 手动操作

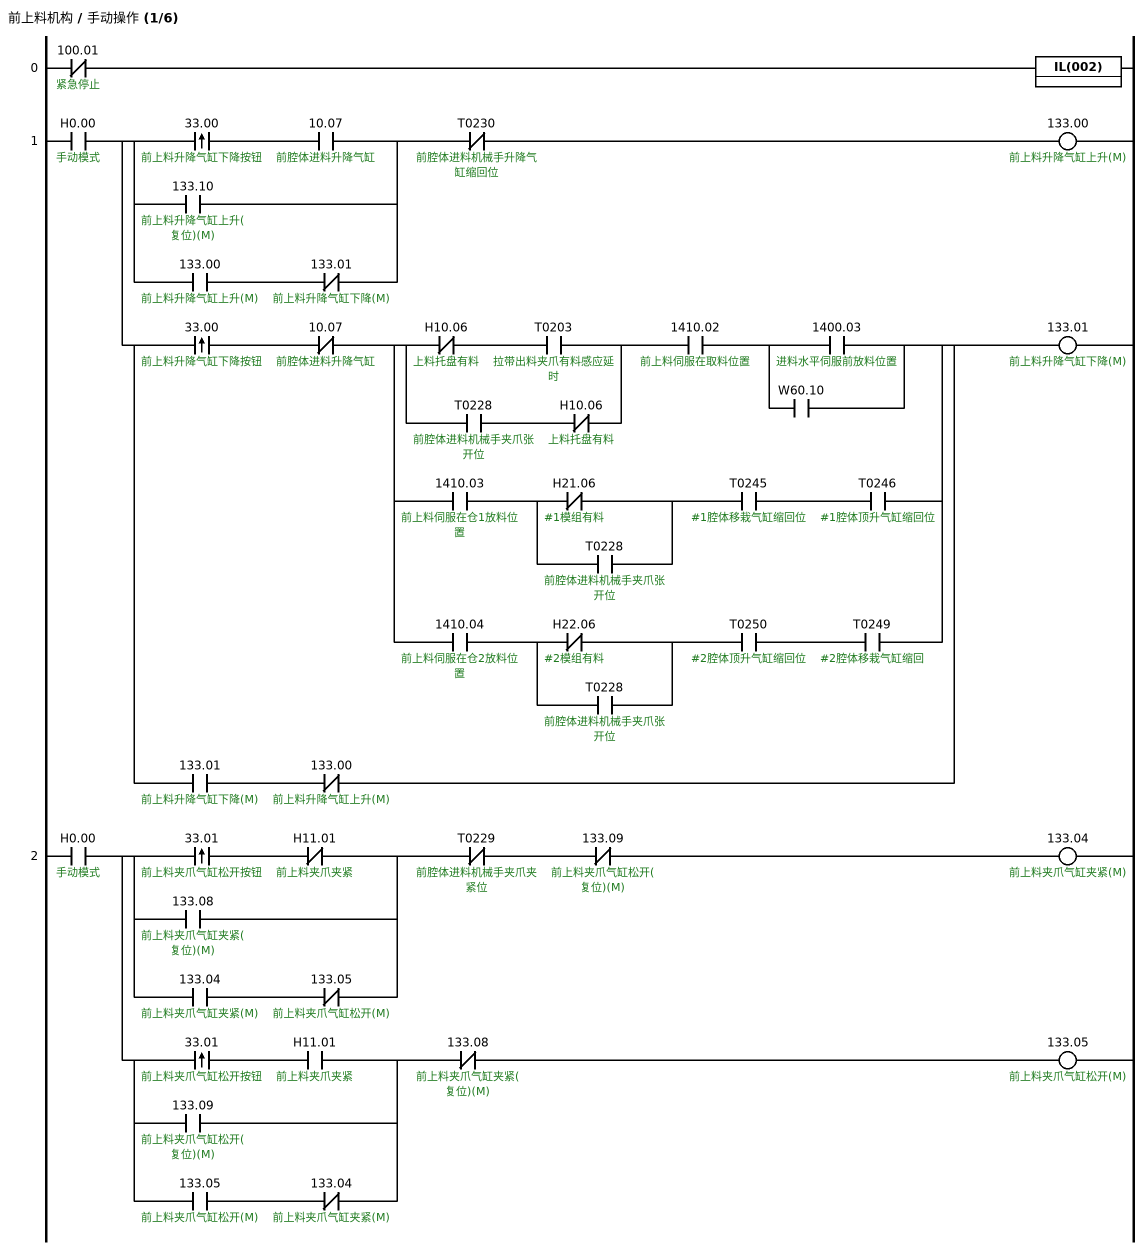
; rung 0
LDNOT 100.01  ; 紧急停止
IL(002)
; rung 1
LD H0.00  ; 手动模式
OUT TR0
@LD 33.00  ; 前上料升降气缸下降按钮
AND 10.07  ; 前腔体进料升降气缸
OR 133.10  ; 前上料升降气缸上升(复位)(M)
LD 133.00  ; 前上料升降气缸上升(M)
ANDNOT 133.01  ; 前上料升降气缸下降(M)
ORLD
ANDLD
ANDNOT T0230  ; 前腔体进料机械手升降气缸缩回位
OUT 133.00  ; 前上料升降气缸上升(M)
LD TR0
@LD 33.00  ; 前上料升降气缸下降按钮
ANDNOT 10.07  ; 前腔体进料升降气缸
LDNOT H10.06  ; 上料托盘有料
AND T0203  ; 拉带出料夹爪有料感应延时
LD T0228  ; 前腔体进料机械手夹爪张开位
ANDNOT H10.06  ; 上料托盘有料
ORLD
AND 1410.02  ; 前上料伺服在取料位置
LD 1400.03  ; 进料水平伺服前放料位置
OR W60.10
ANDLD
LD 1410.03  ; 前上料伺服在仓1放料位置
LDNOT H21.06  ; #1模组有料
OR T0228  ; 前腔体进料机械手夹爪张开位
ANDLD
AND T0245  ; #1腔体移栽气缸缩回位
AND T0246  ; #1腔体顶升气缸缩回位
ORLD
LD 1410.04  ; 前上料伺服在仓2放料位置
LDNOT H22.06  ; #2模组有料
OR T0228  ; 前腔体进料机械手夹爪张开位
ANDLD
AND T0250  ; #2腔体顶升气缸缩回位
AND T0249  ; #2腔体移栽气缸缩回
ORLD
ANDLD
LD 133.01  ; 前上料升降气缸下降(M)
ANDNOT 133.00  ; 前上料升降气缸上升(M)
ORLD
ANDLD
OUT 133.01  ; 前上料升降气缸下降(M)
; rung 2
LD H0.00  ; 手动模式
OUT TR0
@LD 33.01  ; 前上料夹爪气缸松开按钮
ANDNOT H11.01  ; 前上料夹爪夹紧
OR 133.08  ; 前上料夹爪气缸夹紧(复位)(M)
LD 133.04  ; 前上料夹爪气缸夹紧(M)
ANDNOT 133.05  ; 前上料夹爪气缸松开(M)
ORLD
ANDLD
ANDNOT T0229  ; 前腔体进料机械手夹爪夹紧位
ANDNOT 133.09  ; 前上料夹爪气缸松开(复位)(M)
OUT 133.04  ; 前上料夹爪气缸夹紧(M)
LD TR0
@LD 33.01  ; 前上料夹爪气缸松开按钮
AND H11.01  ; 前上料夹爪夹紧
OR 133.09  ; 前上料夹爪气缸松开(复位)(M)
LD 133.05  ; 前上料夹爪气缸松开(M)
ANDNOT 133.04  ; 前上料夹爪气缸夹紧(M)
ORLD
ANDLD
ANDNOT 133.08  ; 前上料夹爪气缸夹紧(复位)(M)
OUT 133.05  ; 前上料夹爪气缸松开(M)

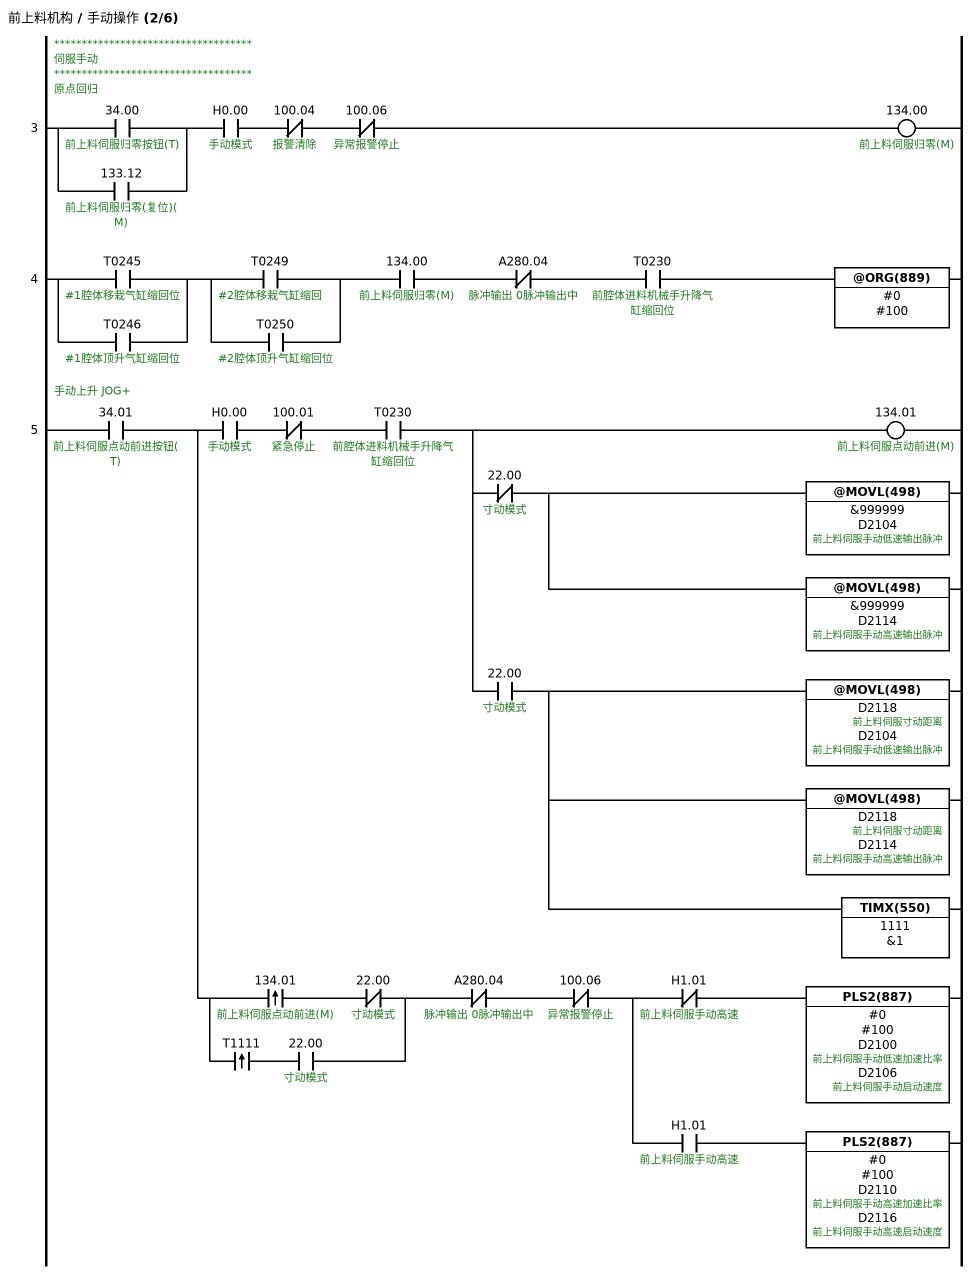
; rung 3: ************************************ / 伺服手动 / ************************************ / 原点回归
LD 34.00  ; 前上料伺服归零按钮(T)
OR 133.12  ; 前上料伺服归零(复位)(M)
AND H0.00  ; 手动模式
ANDNOT 100.04  ; 报警清除
ANDNOT 100.06  ; 异常报警停止
OUT 134.00  ; 前上料伺服归零(M)
; rung 4
LD T0245  ; #1腔体移栽气缸缩回位
OR T0246  ; #1腔体顶升气缸缩回位
LD T0249  ; #2腔体移栽气缸缩回
OR T0250  ; #2腔体顶升气缸缩回位
ANDLD
AND 134.00  ; 前上料伺服归零(M)
ANDNOT A280.04  ; 脉冲输出 0脉冲输出中
AND T0230  ; 前腔体进料机械手升降气缸缩回位
@ORG(889) #0 #100
; rung 5: 手动上升 JOG+
LD 34.01  ; 前上料伺服点动前进按钮(T)
OUT TR0
AND H0.00  ; 手动模式
ANDNOT 100.01  ; 紧急停止
AND T0230  ; 前腔体进料机械手升降气缸缩回位
OUT TR1
OUT 134.01  ; 前上料伺服点动前进(M)
ANDNOT 22.00  ; 寸动模式
@MOVL(498) &999999 D2104  ; 前上料伺服手动低速输出脉冲
@MOVL(498) &999999 D2114  ; 前上料伺服手动高速输出脉冲
LD TR1
AND 22.00  ; 寸动模式
@MOVL(498) D2118 D2104  ; 前上料伺服寸动距离, 前上料伺服手动低速输出脉冲
@MOVL(498) D2118 D2114  ; 前上料伺服寸动距离, 前上料伺服手动高速输出脉冲
TIMX(550) 1111 &1
LD TR0
@LD 134.01  ; 前上料伺服点动前进(M)
ANDNOT 22.00  ; 寸动模式
@LD T1111
AND 22.00  ; 寸动模式
ORLD
ANDLD
ANDNOT A280.04  ; 脉冲输出 0脉冲输出中
ANDNOT 100.06  ; 异常报警停止
OUT TR0
ANDNOT H1.01  ; 前上料伺服手动高速
PLS2(887) #0 #100 D2100 D2106  ; 前上料伺服手动低速加速比率, 前上料伺服手动启动速度
LD TR0
AND H1.01  ; 前上料伺服手动高速
PLS2(887) #0 #100 D2110 D2116  ; 前上料伺服手动高速加速比率, 前上料伺服手动高速启动速度

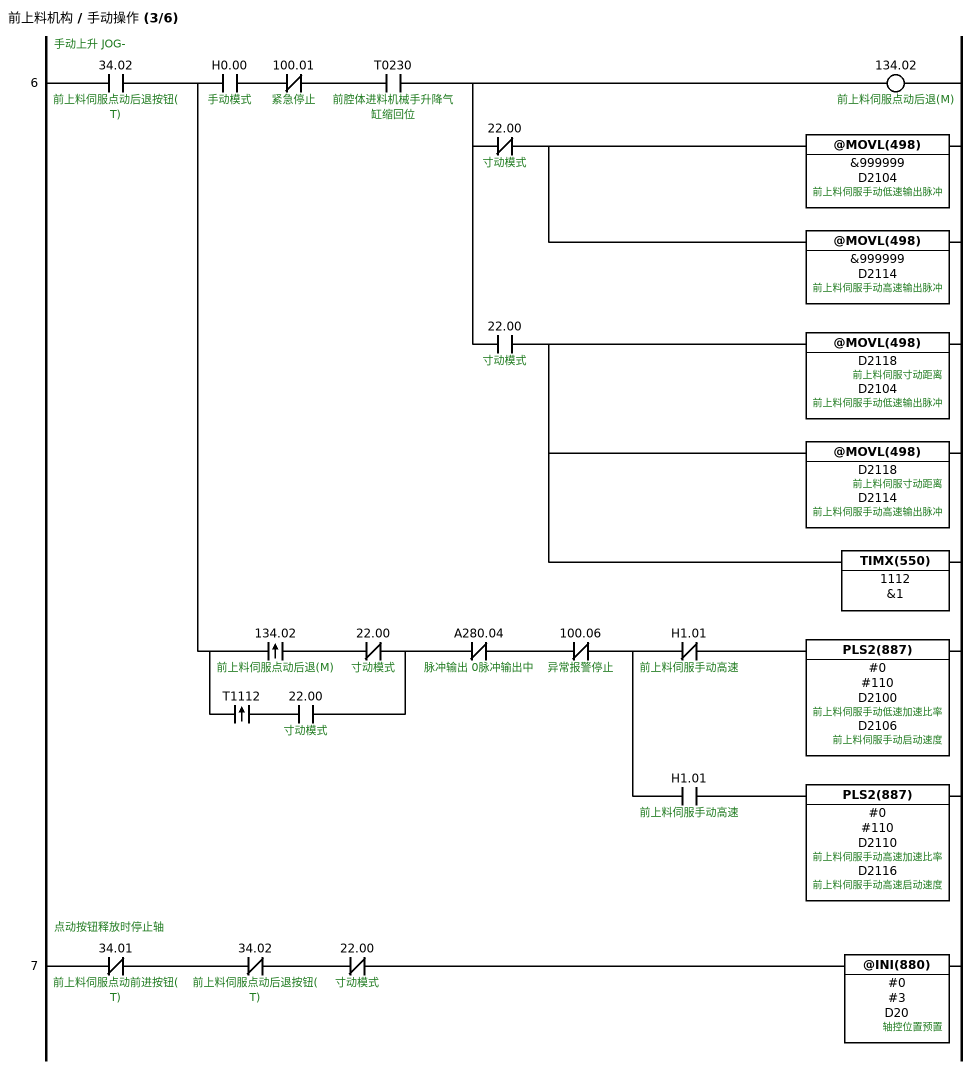
; rung 6: 手动上升 JOG-
LD 34.02  ; 前上料伺服点动后退按钮(T)
OUT TR0
AND H0.00  ; 手动模式
ANDNOT 100.01  ; 紧急停止
AND T0230  ; 前腔体进料机械手升降气缸缩回位
OUT TR1
OUT 134.02  ; 前上料伺服点动后退(M)
ANDNOT 22.00  ; 寸动模式
@MOVL(498) &999999 D2104  ; 前上料伺服手动低速输出脉冲
@MOVL(498) &999999 D2114  ; 前上料伺服手动高速输出脉冲
LD TR1
AND 22.00  ; 寸动模式
@MOVL(498) D2118 D2104  ; 前上料伺服寸动距离, 前上料伺服手动低速输出脉冲
@MOVL(498) D2118 D2114  ; 前上料伺服寸动距离, 前上料伺服手动高速输出脉冲
TIMX(550) 1112 &1
LD TR0
@LD 134.02  ; 前上料伺服点动后退(M)
ANDNOT 22.00  ; 寸动模式
@LD T1112
AND 22.00  ; 寸动模式
ORLD
ANDLD
ANDNOT A280.04  ; 脉冲输出 0脉冲输出中
ANDNOT 100.06  ; 异常报警停止
OUT TR0
ANDNOT H1.01  ; 前上料伺服手动高速
PLS2(887) #0 #110 D2100 D2106  ; 前上料伺服手动低速加速比率, 前上料伺服手动启动速度
LD TR0
AND H1.01  ; 前上料伺服手动高速
PLS2(887) #0 #110 D2110 D2116  ; 前上料伺服手动高速加速比率, 前上料伺服手动高速启动速度
; rung 7: 点动按钮释放时停止轴
LDNOT 34.01  ; 前上料伺服点动前进按钮(T)
ANDNOT 34.02  ; 前上料伺服点动后退按钮(T)
ANDNOT 22.00  ; 寸动模式
@INI(880) #0 #3 D20  ; 轴控位置预置

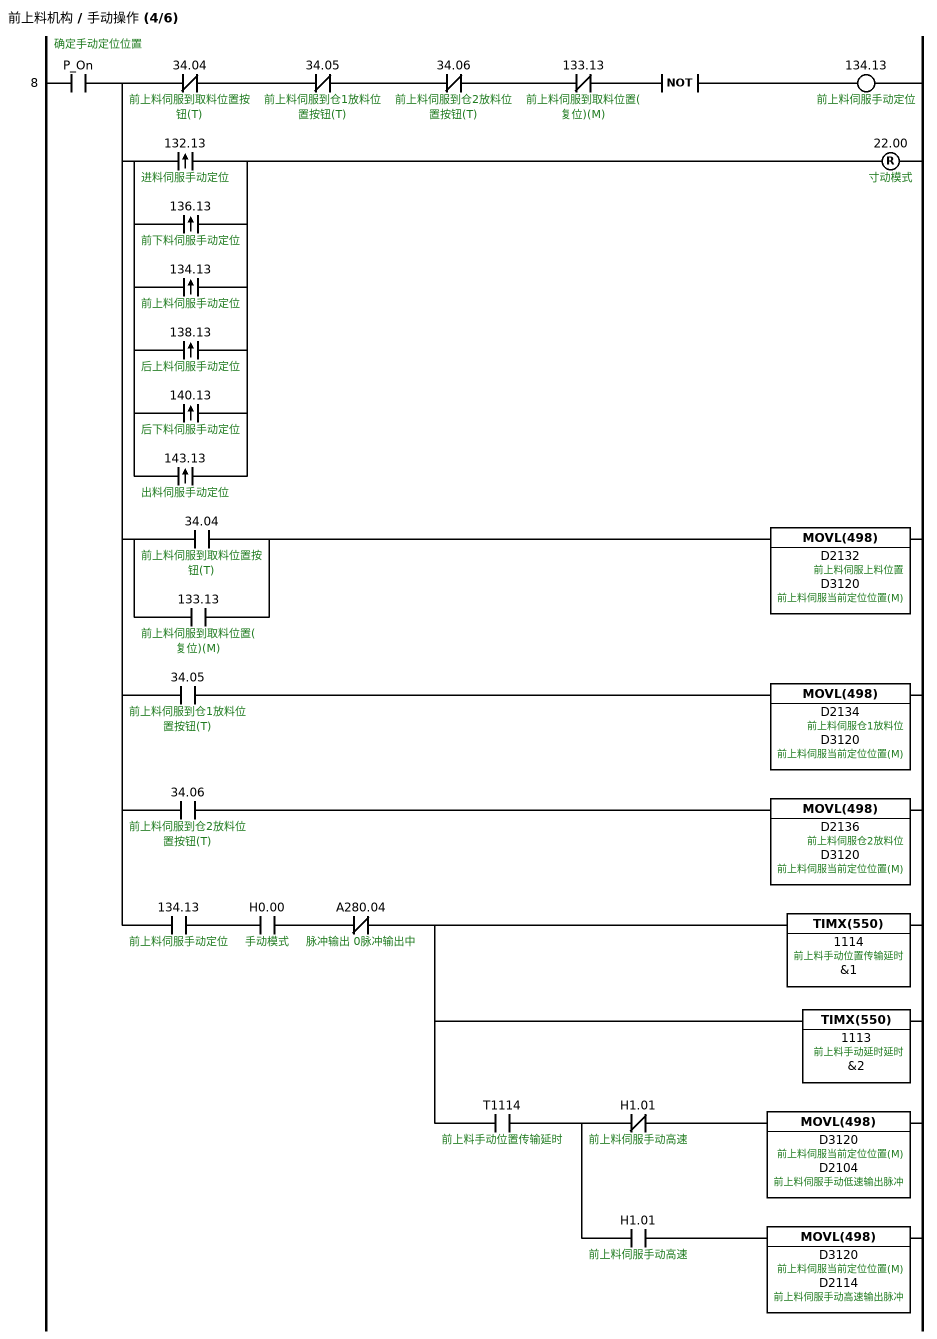
; rung 8: 确定手动定位位置
LD P_On
OUT TR0
ANDNOT 34.04  ; 前上料伺服到取料位置按钮(T)
ANDNOT 34.05  ; 前上料伺服到仓1放料位置按钮(T)
ANDNOT 34.06  ; 前上料伺服到仓2放料位置按钮(T)
ANDNOT 133.13  ; 前上料伺服到取料位置(复位)(M)
NOT(520)
OUT 134.13  ; 前上料伺服手动定位
LD TR0
@LD 132.13  ; 进料伺服手动定位
@OR 136.13  ; 前下料伺服手动定位
@OR 134.13  ; 前上料伺服手动定位
@OR 138.13  ; 后上料伺服手动定位
@OR 140.13  ; 后下料伺服手动定位
@OR 143.13  ; 出料伺服手动定位
ANDLD
RSET 22.00  ; 寸动模式
LD TR0
LD 34.04  ; 前上料伺服到取料位置按钮(T)
OR 133.13  ; 前上料伺服到取料位置(复位)(M)
ANDLD
MOVL(498) D2132 D3120  ; 前上料伺服上料位置, 前上料伺服当前定位位置(M)
LD TR0
AND 34.05  ; 前上料伺服到仓1放料位置按钮(T)
MOVL(498) D2134 D3120  ; 前上料伺服仓1放料位, 前上料伺服当前定位位置(M)
LD TR0
AND 34.06  ; 前上料伺服到仓2放料位置按钮(T)
MOVL(498) D2136 D3120  ; 前上料伺服仓2放料位, 前上料伺服当前定位位置(M)
LD TR0
AND 134.13  ; 前上料伺服手动定位
AND H0.00  ; 手动模式
ANDNOT A280.04  ; 脉冲输出 0脉冲输出中
TIMX(550) 1114 &1  ; 前上料手动位置传输延时
TIMX(550) 1113 &2  ; 前上料手动延时延时
AND T1114  ; 前上料手动位置传输延时
OUT TR0
ANDNOT H1.01  ; 前上料伺服手动高速
MOVL(498) D3120 D2104  ; 前上料伺服当前定位位置(M), 前上料伺服手动低速输出脉冲
LD TR0
AND H1.01  ; 前上料伺服手动高速
MOVL(498) D3120 D2114  ; 前上料伺服当前定位位置(M), 前上料伺服手动高速输出脉冲

